INTERFACE I_Power

METHOD Power
VAR_INPUT
    Enable	: BOOL;
    Enable_Positive	: BOOL;
    Enable_Negative	: BOOL;
    Override	: LREAL ;
    BufferMode	: MC_BufferMode;
END_VAR
END_METHOD

PROPERTY PowerActive : BOOL
GET
END_GET
END_PROPERTY

PROPERTY PowerEnable : BOOL
SET
END_SET
END_PROPERTY

PROPERTY PowerEnableNegative : BOOL
SET
END_SET
END_PROPERTY

PROPERTY PowerEnablePositive : BOOL
SET
END_SET
END_PROPERTY

PROPERTY PowerError : BOOL
GET
END_GET
END_PROPERTY

PROPERTY PowerErrorID : UDINT
GET
END_GET
END_PROPERTY

PROPERTY PowerIsEnabled : BOOL
GET
END_GET
END_PROPERTY

PROPERTY PowerOverride : LREAL
SET
END_SET
END_PROPERTY

END_INTERFACE

(* stored: Version 1.1.0.1
   Itf I_Power: Id {3e27e6e8-6685-424d-9ead-eda513d1c175}
   Method Power: Id {6ec5953f-7853-4ae8-b7bf-ca6c5f20defd}
   Property PowerActive: Id {20b72d22-0b79-4e66-8e59-11a346450f29}
   Get Get: Id {f893a206-91ba-4636-8483-e8eab88dcb57}
   Property PowerEnable: Id {1110da7f-53f9-4d9e-acd2-6779b9ac57bb}
   Set Set: Id {68ce8530-0b4e-49b2-b142-87874089ade1}
   Property PowerEnableNegative: Id {f4468a5f-99c2-41ef-8494-82f11d6af19e}
   Set Set: Id {325c8bbd-cb6f-445c-bdde-af74df7c86c0}
   Property PowerEnablePositive: Id {a7e67244-44ea-4632-8730-f811e553e6c7}
   Set Set: Id {665a290f-0612-4dd5-8ddf-d027af35e44f}
   Property PowerError: Id {6604d428-f1f1-4c20-a8b9-dc8f79a70991}
   Get Get: Id {b3c2d465-f80b-44c6-b7a9-42c9686181fe}
   Property PowerErrorID: Id {ab8e474d-c533-46cf-82e5-024666820951}
   Get Get: Id {640c781c-4181-42bc-8810-58d857789713}
   Property PowerIsEnabled: Id {51943bc5-fd82-4d37-a623-d1f89afd6f2e}
   Get Get: Id {f6f920c1-2a15-45fb-99e2-22914eacf6cf}
   Property PowerOverride: Id {05600e99-3607-4f22-b5d2-f539e7fc2cd3}
   Set Set: Id {d6569857-2f15-4c83-a4a1-ba171e758562} *)
